FUNCTION FC_4strConcat : T_DEFAULT_STR		// Concatenates 4 strings
VAR_INPUT
	iStr1:		T_DEFAULT_STR;
	iStr2:		T_DEFAULT_STR;
	iStr3:		T_DEFAULT_STR;
	iStr4:		T_DEFAULT_STR;
END_VAR

FC_4strConcat := CONCAT(FC_3strConcat(iStr1, iStr2, iStr3), iStr4);

END_FUNCTION

(* stored: Version 1.1.0.1, ProductVersion 3.1.4026.18
   POU FC_4strConcat: Id {9204972f-038a-499d-bd44-a70f01cbf2d6}, SpecialFunc None *)
